FUNCTION "LEN_LS_1" : UInt
{ S7_Optimized_Access := 'TRUE' }
VERSION : 0.1
   VAR_IN_OUT
      IN : "t_LString";
   END_VAR


BEGIN
	#LEN_LS_1 := #IN.Len;
END_FUNCTION

